VAR_GLOBAL
	arr AT%MW0: ARRAY [0..2] OF WORD;
END_VAR

(* stored: Version 1.1.0.1, ProductVersion 3.1.0.38
   GVL GVL: Id {c048432b-d782-49ea-a20f-cf84ef79fc78} *)
